TYPE VECTOR_3 :
STRUCT
	X : REAL;
	Y : REAL;
	Z : REAL;
END_STRUCT
END_TYPE

(* stored: Version 1.1.0.1, ProductVersion 3.1.4024.9
   DUT VECTOR_3: Id {a1f7b061-0062-4dd4-bc0f-65a269a87f69} *)
